FUNCTION_BLOCK ST_DEL_CONN (* Deletes an event or data connection between two FB instances *)
  (* Standard: 61499-1; Classification: Reconfiguration; Function: Deletes Connection; Type: Structural Service *)
  (* Version 1.0, 2012-06-01, EG, 4DIAC-Consortium *)
  (* Compiler Cpp GNU GCC >3.0 *)
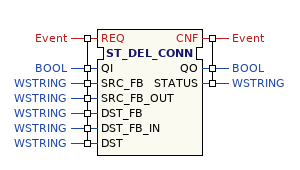
  EVENT_INPUT
    REQ WITH SRC_FB, SRC_FB_OUT, DST_FB, DST_FB_IN, DST, QI; (* Event to require deletion of a connection *)
  END_EVENT
  EVENT_OUTPUT
    CNF WITH STATUS, QO; (* Event to confirm that the connection has been deleted *)
  END_EVENT
  VAR_INPUT
    QI : BOOL; (* Event Input Qualifier *)
    SRC_FB : WSTRING; (* Reference to Source FB instance *)
    SRC_FB_OUT : WSTRING; (* Reference to Source FB instance Event/Data-Output *)
    DST_FB : WSTRING; (* Reference to Destination FB instance *)
    DST_FB_IN : WSTRING; (* Reference to Destination FB instance Event/Data-Input *)
    DST : WSTRING; (* Destination where the connection has to be deleted (Syntax: ResourceName) *)
  END_VAR
  VAR_OUTPUT
    QO : BOOL; (* Event Output Qualifier *)
    STATUS : WSTRING; (* Service Status: RDY, NO_SUCH_OBJECT *)
  END_VAR
  SERVICE APPLICATION/RESOURCE (* Deletes an event or data connection between two FB instances *)
    SEQUENCE normal_establishment
      APPLICATION.INIT+() -> APPLICATION.INITO+();
    END_SEQUENCE
    SEQUENCE unsuccessful_establishment
      APPLICATION.INIT+() -> APPLICATION.INITO-();
    END_SEQUENCE
    SEQUENCE request_confirm
      APPLICATION.REQ+() -> APPLICATION.CNF+();
    END_SEQUENCE
    SEQUENCE request_inhibited
      APPLICATION.REQ-() -> APPLICATION.CNF-();
    END_SEQUENCE
    SEQUENCE request_error
      APPLICATION.REQ+() -> APPLICATION.CNF-();
    END_SEQUENCE
    SEQUENCE application_initiated_termination
      APPLICATION.INIT-() -> APPLICATION.INITO-();
    END_SEQUENCE
    SEQUENCE resource_initiated_termination
      -> APPLICATION.INITO-();
    END_SEQUENCE
  END_SERVICE
END_FUNCTION_BLOCK
